FUNCTION_BLOCK Motor
VAR_INPUT
END_VAR
VAR_OUTPUT
END_VAR
VAR
	wDeviceAddress : WORD;
	rSpeedActual : REAL;
	rTorqueActual: REAL;
	rCurrentActual : REAL;
	rSpeedSetpoint : REAL;
	rTorqueSetpoint : REAL;
	bPowerStatus : BOOL;
	wErrorStatus : WORD;
END_VAR

PROPERTY PUBLIC currentActual : REAL
GET
currentActual := rCurrentActual;
END_GET
END_PROPERTY

PROPERTY PUBLIC errorStatus : WORD
GET
errorStatus := wErrorStatus;
END_GET
END_PROPERTY

METHOD FB_init : BOOL
VAR_INPUT
	bInitRetains : BOOL; // if TRUE, the retain variables are initialized (warm start / cold start)
	bInCopyCode : BOOL;  // if TRUE, the instance afterwards gets moved into the copy code (online change)
END_VAR
END_METHOD

PROPERTY PUBLIC powerStatus : BOOL
GET
powerStatus := bPowerStatus;
END_GET
END_PROPERTY

METHOD PUBLIC setSpeedSetpoint : BOOL
VAR_INPUT
END_VAR
END_METHOD

METHOD PUBLIC setTorqueSetpoint : BOOL
VAR_INPUT
END_VAR
END_METHOD

PROPERTY PUBLIC speedActual : REAL
GET
speedActual := rSpeedActual;
END_GET
END_PROPERTY

METHOD start : BOOL
VAR_INPUT
END_VAR
END_METHOD

METHOD stop : BOOL
VAR_INPUT
END_VAR
END_METHOD

PROPERTY PUBLIC torqueActual : REAL
GET
torqueActual := rTorqueActual;
END_GET
END_PROPERTY

END_FUNCTION_BLOCK

(* stored: Version 1.1.0.1, ProductVersion 3.1.4024.12
   POU Motor: Id {9e201c52-51a5-4466-a32f-9add5cad1d22}, SpecialFunc None
   Property currentActual: Id {701a1092-a4e5-492f-bd19-0634763c5c80}
   Get Get: Id {c4383f64-d485-43a2-8306-9afc637da0ab}
   Property errorStatus: Id {e3900296-98d3-4e55-82fb-8730b9dcfdbd}
   Get Get: Id {10296193-d52c-4171-9ff8-73751dab9d1b}
   Method FB_init: Id {8492f597-30a8-4e60-bad6-32c194051611}
   Property powerStatus: Id {871ea45a-1a3c-4dad-8f01-1ccb0a84c3af}
   Get Get: Id {55aefbc5-50ff-4152-9691-a098436216ff}
   Method setSpeedSetpoint: Id {8ff61fd8-1855-4e7d-9484-bd5d274d55cb}
   Method setTorqueSetpoint: Id {7c9d246f-b088-41e7-bd54-9eb802ad7907}
   Property speedActual: Id {ae7bd87f-c844-4ac9-9ef2-13638a6e2282}
   Get Get: Id {6c1d829d-a8ae-4c9b-9edf-463187e727a0}
   Method start: Id {decf84df-c562-4530-8600-dd47fe5d0e03}
   Method stop: Id {8be7300a-91cb-4938-a75f-8a2aef468905}
   Property torqueActual: Id {c52aedf7-edde-4e34-8d7d-b672f91bce09}
   Get Get: Id {806f4ae0-04f0-4883-a618-5835db72cf62} *)
